TYPE st_OperatingPoint :
STRUCT
	OperatingMode	:	eHeatpumpMode;
	Setpoint		:	REAL;
END_STRUCT
END_TYPE

(* stored: Version 1.1.0.1, ProductVersion 3.1.4024.12
   DUT st_OperatingPoint: Id {c3cf3b58-5238-4d23-9ded-465a43b916e0} *)
